FUNCTION_BLOCK FB_ThNTZ_Logik
VAR_IN_OUT
	Steuerung	: ST_ThNTZ_Steuerung;
	Zustand		: ST_ThNTZ_Zustand;
END_VAR
VAR_INPUT
	Parameter	: ST_ThNTZ_Parameter;
END_VAR
VAR_OUTPUT
END_VAR
VAR
END_VAR

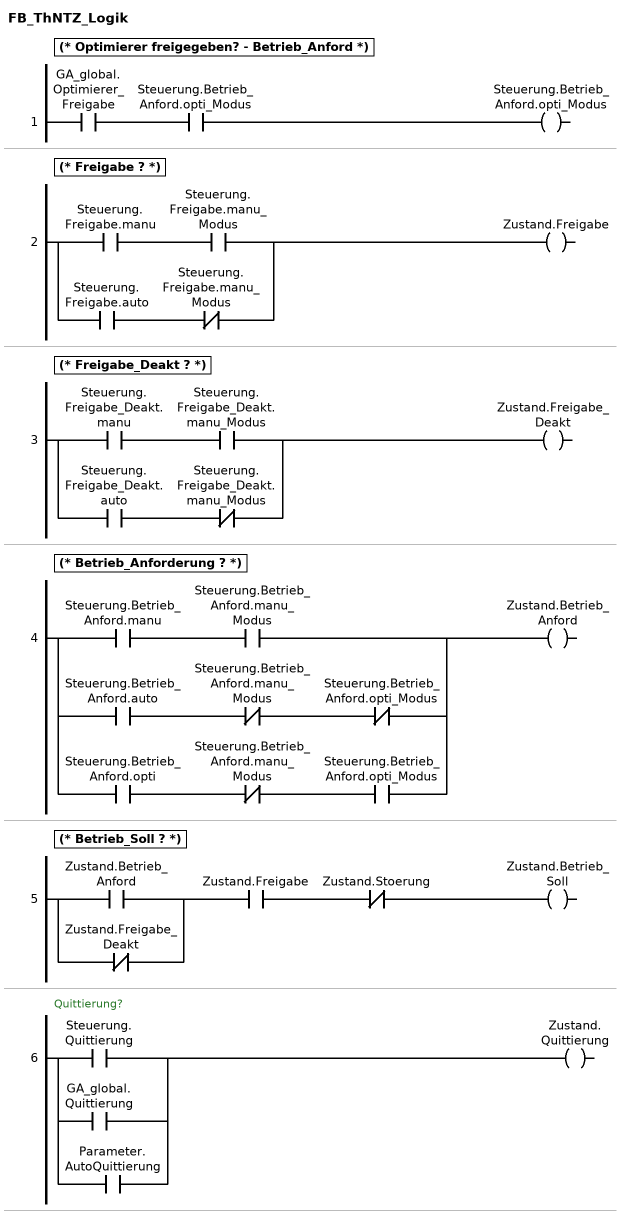
// NETWORK 1
// label: (* Optimierer freigegeben? - Betrieb_Anford *)
Steuerung.Betrieb_Anford.opti_Modus := GA_global.Optimierer_Freigabe AND Steuerung.Betrieb_Anford.opti_Modus;

// NETWORK 2
// label: (* Freigabe ? *)
Zustand.Freigabe := Steuerung.Freigabe.manu AND Steuerung.Freigabe.manu_Modus OR Steuerung.Freigabe.auto AND NOT Steuerung.Freigabe.manu_Modus;

// NETWORK 3
// label: (* Freigabe_Deakt ? *)
Zustand.Freigabe_Deakt := Steuerung.Freigabe_Deakt.manu AND Steuerung.Freigabe_Deakt.manu_Modus OR Steuerung.Freigabe_Deakt.auto AND NOT Steuerung.Freigabe_Deakt.manu_Modus;

// NETWORK 4
// label: (* Betrieb_Anforderung ? *)
Zustand.Betrieb_Anford := Steuerung.Betrieb_Anford.manu AND Steuerung.Betrieb_Anford.manu_Modus OR Steuerung.Betrieb_Anford.auto AND NOT Steuerung.Betrieb_Anford.manu_Modus AND NOT Steuerung.Betrieb_Anford.opti_Modus OR Steuerung.Betrieb_Anford.opti AND NOT Steuerung.Betrieb_Anford.manu_Modus AND Steuerung.Betrieb_Anford.opti_Modus;

// NETWORK 5
// label: (* Betrieb_Soll ? *)
Zustand.Betrieb_Soll := (Zustand.Betrieb_Anford OR NOT Zustand.Freigabe_Deakt) AND Zustand.Freigabe AND NOT Zustand.Stoerung;

// NETWORK 6
// Quittierung?
Zustand.Quittierung := Steuerung.Quittierung OR GA_global.Quittierung OR Parameter.AutoQuittierung;

END_FUNCTION_BLOCK

(* stored: Version 1.1.0.1, ProductVersion 3.1.4024.9
   POU FB_ThNTZ_Logik: Id {5535e56b-f87d-460d-9f98-532a92b3f162}, SpecialFunc None *)
